PROGRAM prg_DraaiRichtingMotor
VAR
END_VAR

END_PROGRAM

(* stored: Version 1.1.0.1, ProductVersion 3.1.4024.15
   POU prg_DraaiRichtingMotor: Id {52597bfd-aa8a-4647-945c-0d4f5bed4876}, SpecialFunc None *)
